// TIA Portal project "esContatore" (V16)
// esercizio autoritenuta

(* hardware
DEVICE "S7-1200 station_1"  S7-1200 Station
   slot 0: "Telaio di montaggio_0"  S7-1200 Rack  Rack  V1.0
   slot 1: "PLC_1"  CPU 1215C DC/DC/Rly  6ES7 215-1HG40-0XB0  V4.4
*)

// ===== PLC "PLC_1"  CPU 1215C DC/DC/Rly =====

VAR_GLOBAL   // PLC tag table "Tabella delle variabili standard"
   "Marcia" AT %I1.0 : Bool;   // Commento su marcia
   "Emergenza" AT %I0.7 : Bool;
   "Start" AT %I1.1 : Bool;
   "Arresto" AT %I1.2 : Bool;
   "Macchina On" AT %M0.0 : Bool;   // Macchina merkel accesa
   "Avanti" AT %Q0.0 : Bool;
   "Indietro" AT %Q0.1 : Bool;
   "Spia macchina accesa" AT %Q0.6 : Bool;
   "Fotocellula1" AT %I0.0 : Bool;
   "Fotocellula2" AT %I0.1 : Bool;
   "Spia avanti" AT %Q0.7 : Bool;
   "Spia indietro" AT %Q1.0 : Bool;
   "arrivato" AT %M0.1 : Bool;
   "ritornato" AT %M0.2 : Bool;
   "fine" AT %M0.3 : Bool;
   "reset" AT %M0.4 : Bool;
END_VAR

// folder: System blocks/Program resources

DATA_BLOCK "IEC_Counter_0_DB"   // DB1
{ S7_Optimized_Access := 'TRUE' }
AUTHOR : Simatic
FAMILY : IEC
NAME : CNTR
VERSION : 1.0
// stored: InstanceOfName IEC_COUNTER
"IEC_COUNTER"
BEGIN
END_DATA_BLOCK

// folder: (top level)

ORGANIZATION_BLOCK "Main"   // OB1, LAD, ProgramCycle
TITLE = "Main Program Sweep (Cycle)" / Macchina1
{ S7_Optimized_Access := 'TRUE' }
VERSION : 0.1
// Esercizio contatore
   VAR_INPUT
      Initial_Call : Bool;   // Initial call of this OB
      Remanence : Bool;   // =True, if remanent data are available
   END_VAR
BEGIN

REGION Network 1: Gestione della macchina accesa
   // Marcia (m) - Emergenza(e)
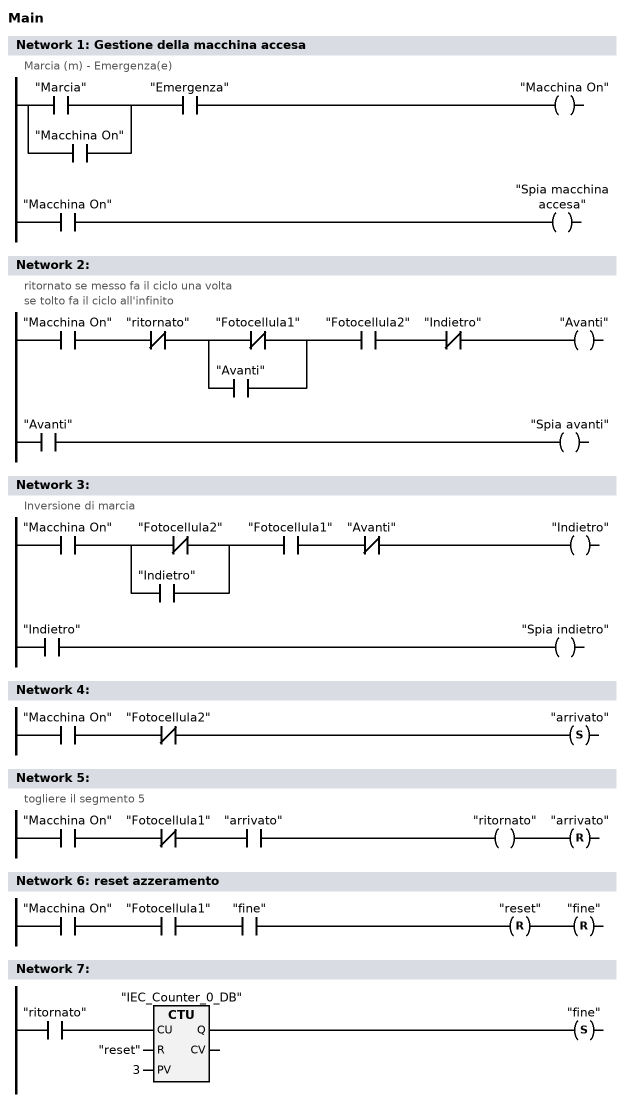
   RUNG wire#powerrail
      Contact( "Marcia" )
      wire#w1
      Contact( "Emergenza" )
      Coil( "Macchina On" )
   END_RUNG
   RUNG wire#powerrail
      Contact( "Macchina On" )
   END_RUNG wire#w1
   RUNG wire#powerrail
      Contact( "Macchina On" )
      Coil( "Spia macchina accesa" )
   END_RUNG
   // the same network as SCL:
   "Macchina On" := ("Marcia" OR "Macchina On") AND "Emergenza";
   "Spia macchina accesa" := "Macchina On";
END_REGION

REGION Network 2
   // ritornato se messo fa il ciclo una volta 
   // se tolto fa il ciclo all'infinito
   RUNG wire#powerrail
      Contact( "Macchina On" )
      I_Contact( "ritornato" )
      wire#w1
      I_Contact( "Fotocellula1" )
      wire#w2
      Contact( "Fotocellula2" )
      I_Contact( "Indietro" )
      Coil( "Avanti" )
   END_RUNG
   RUNG wire#w1
      Contact( "Avanti" )
   END_RUNG wire#w2
   RUNG wire#powerrail
      Contact( "Avanti" )
      Coil( "Spia avanti" )
   END_RUNG
   // the same network as SCL:
   "Avanti" := "Macchina On" AND NOT "ritornato" AND (NOT "Fotocellula1" OR "Avanti") AND "Fotocellula2" AND NOT "Indietro";
   "Spia avanti" := "Avanti";
END_REGION

REGION Network 3
   // Inversione di marcia
   RUNG wire#powerrail
      Contact( "Macchina On" )
      wire#w1
      I_Contact( "Fotocellula2" )
      wire#w2
      Contact( "Fotocellula1" )
      I_Contact( "Avanti" )
      Coil( "Indietro" )
   END_RUNG
   RUNG wire#w1
      Contact( "Indietro" )
   END_RUNG wire#w2
   RUNG wire#powerrail
      Contact( "Indietro" )
      Coil( "Spia indietro" )
   END_RUNG
   // the same network as SCL:
   "Indietro" := "Macchina On" AND (NOT "Fotocellula2" OR "Indietro") AND "Fotocellula1" AND NOT "Avanti";
   "Spia indietro" := "Indietro";
END_REGION

REGION Network 4
   RUNG wire#powerrail
      Contact( "Macchina On" )
      I_Contact( "Fotocellula2" )
      S_Coil( "arrivato" )
   END_RUNG
   // the same network as SCL:
   IF "Macchina On" AND NOT "Fotocellula2" THEN "arrivato" := TRUE; END_IF;
END_REGION

REGION Network 5
   // togliere il segmento 5
   RUNG wire#powerrail
      Contact( "Macchina On" )
      I_Contact( "Fotocellula1" )
      Contact( "arrivato" )
      Coil( "ritornato" )
      R_Coil( "arrivato" )
   END_RUNG
   // the same network as SCL:
   "ritornato" := "Macchina On" AND NOT "Fotocellula1" AND "arrivato";
   IF "ritornato" THEN "arrivato" := FALSE; END_IF;
END_REGION

REGION Network 6: reset azzeramento
   RUNG wire#powerrail
      Contact( "Macchina On" )
      Contact( "Fotocellula1" )
      Contact( "fine" )
      R_Coil( "reset" )
      R_Coil( "fine" )
   END_RUNG
   // the same network as SCL:
   IF "Macchina On" AND "Fotocellula1" AND "fine" THEN
       "reset" := FALSE;
       "fine" := FALSE;
   END_IF;
END_REGION

REGION Network 7
   "IEC_Counter_0_DB".CTU(CU := "ritornato", R := "reset", PV := 3);
   IF "IEC_Counter_0_DB".Q THEN "fine" := TRUE; END_IF;
END_REGION
END_ORGANIZATION_BLOCK